Staubli VAL3: Prog1.dtx

public frame fReference = {fatherId=world[0]}
public jointRx jPark = {j3=90, j5=90}
public jointRx jJoint
public mdesc mNomSpeed = {blend=off}
public mdesc mSpeed[0]
public num nTraj
num nTimeStop
num nTimeStart
num nMode
num nEtat
public pointRx pPoint[2]
  [0] = {x=1374.251, y=-500, z=294.734, rx=158.451, ry=10.915, rz=133.958, shoulder=lefty, elbow=epositive, wrist=wpositive, fatherId=fReference[0]}
  [1] = {x=1374.251, y=500, z=294.734, rx=-168.326, ry=14.136, rz=131.26, shoulder=lefty, elbow=epositive, wrist=wpositive, fatherId=fReference[0]}
public tool tTool = {x=-55.6, y=-198.63, z=-982.79, fatherId=flange[0], ioLink=valve1}
